// TIA Portal V17 export
// export: Created 2025-03-10T12:16:06.6393818Z, ExportSetting WithDefaults, DisplayName Totally Integrated Automation Portal, DisplayVersion V17 Update 8, DisplayName TIA Portal Openness, DisplayVersion V17 Update 8, DisplayName TIA Portal Version Control Interface, DisplayVersion V17, DisplayName SINAMICS Startdrive Advanced, DisplayVersion V17 SP2, DisplayName SINAMICS Startdrive G110M, G120, G120C, G120D, G120P, G115D, DisplayVersion V17 SP2, DisplayName SINAMICS Startdrive G130, G150, S120, S150, SINAMICS MV, S210, DisplayVersion V17 SP2, DisplayName STEP 7 Professional, DisplayVersion V17 Update 8, DisplayName SINUMERIK ONE STEP 7 Toolbox, DisplayVersion V17 Update 12, DisplayName SINUMERIK 840D sl STEP 7 Toolbox, DisplayVersion V17 Update 12, DisplayName STEP 7 Safety, DisplayVersion V17 Update 6, DisplayName WinCC Advanced, DisplayVersion V17 Update 8
DATA_BLOCK "DB136_CLADDING_SPINDLE_C14"   // DB136
{ DB_Accessible_From_OPC_UA := 'FALSE' }
AUTHOR : ETXETAR
VERSION : 1.0
// stored: AutoNumber false, DBAccessibleFromOPCUA false, DBAccessibleFromWebserver true, InstanceOfName FB31_SPINDLE, InstanceOfType FB
"FB31_SPINDLE"
   // VAR_INPUT
   //    OPTIONS_0 : Byte;
   //    OPTIONS_1 : Byte;
   //    SAFETY_BYPASS : Bool;
   //    OPTIMIZATION_BYPASS : Bool;
   //    RPMS_REACHED : Bool;
   //    BELT_BROKEN : Bool;
   //    COOLING_SYS_IN_SERVICE : Bool;
   //    MQL_HP_IN_SERVICE : Bool;
   //    TEMPERATURE_SENSOR : Word;
   //    TEMPERATURE_SENSOR_PTC : Bool;
   //    VPM_READY : Bool;
   //    ENABLE : Bool;
   //    FEED_HOLD_COND : Bool;
   //    UNIT_SEQ_RUNNING : Bool;
   //    SAFE_ENABLED : Bool;
   //    TEST_STOP_INTERNAL_PULSES : Bool;
   //    FEED_OVERRIDE : Byte;
   //    SPINDLE_OVERRIDE : Byte;
   //    HMI_SP_SELECTED : Bool;
   //    HMI_REQ_LINE : Bool;
   //    CHANNEL_M3 : Bool;
   //    CHANNEL_M300 : Bool;
   //    M_VERIFY_CLAMP_F1 : Bool;
   //    M_VERIFY_CLAMP_F2 : Bool;
   //    SP_CLAMP : Bool;
   //    SP_CLAMPED : Bool;
   //    SP_CLAMPED_WITH_TOOL : Bool;
   //    HARDWARE_ENABLE : Bool;
   //    TOOL_CHANGE_POS : Bool;
   //    FIXTURE_1_PART_OK : Bool;
   //    FIXTURE_2_PART_OK : Bool;
   //    READ_POS : DWord;
   //    UNIT_ALARM : UInt;
   //    STATION_ALARM : UInt;
   //    DESELECT_SPINDLE_STO : Bool;
   // END_VAR
   // VAR_OUTPUT
   //    DELAYED_ENABLE : Bool;
   //    FEED_HOLD_CONDITIONS : Bool;
   //    FEED_HOLD_CONDITIONS_HMI : Bool;
   //    SP_DESELECTED : Bool;
   //    SPEED_NOT_REACHED_ALARM : Bool;
   //    BELT_BROKEN_ALARM : Bool;
   //    COOLING_ALARM : Bool;
   //    MQL_HP_ALARM : Bool;
   //    HIGH_TEMP_ALARM : Bool;
   //    HIGH_TEMP_PTC_ALARM : Bool;
   //    VPM_READY_ALARM : Bool;
   //    HIGH_TEMP_PREALM : Bool;
   //    SPINDLE_POS : Real;
   //    HMI_MOTION_EXECUTABILITY_LEFT : Bool;
   //    HMI_MOTION_EXECUTABILITY_RIGHT : Bool;
   //    HMI_MOTION_END_POS_LEFT : Bool;
   //    HMI_MOTION_END_POS_RIGHT : Bool;
   // END_VAR
   // VAR_IN_OUT
   //    SpindleDB : "LBP_typeAxisX";
   // END_VAR
   // VAR RETAIN
   //    SP : "SPINDLE";
   //    SP_TEMPERATURE : Real;
   //    TEMP_MUL_VAL { S7_SetPoint := 'True'} : Real;
   //    TEMP_DIV_VAL { S7_SetPoint := 'True'} : Real;
   //    TEMP_SUB_VAL { S7_SetPoint := 'True'} : Real;
   //    TEMP_PREALARM_VAL { S7_SetPoint := 'True'} : Real;
   //    TEMP_ALARM_VAL { S7_SetPoint := 'True'} : Real;
   //    WARNING_GONE { S7_SetPoint := 'True'} : Bool;
   //    TIMER_ENABLE_PULSE { S7_SetPoint := 'True'} : TOF_TIME;
   //    TIMER_DELETE_DIST_TO_GO { S7_SetPoint := 'True'} : TON_TIME;
   //    TIMER_SPEED_NOT_REACHED { S7_SetPoint := 'True'} : TOF_TIME;
   //    TIMER_BELT_BROKEN_ALARM { S7_SetPoint := 'True'} : TON_TIME;
   //    TIMER_MQL_HP_FAULT { S7_SetPoint := 'True'} : TON_TIME;
   //    TIMER_COMMAND_JOG_PLUS { S7_SetPoint := 'True'} : TON_TIME;
   //    SAFETY_POSITIONS { S7_SetPoint := 'True'} : "FB33_SAFETY_POSITIONS";
   // END_VAR
BEGIN
END_DATA_BLOCK
